{attribute addProperty BoxType "APS1003-5000-0016"}
{attribute addProperty Id "FB_InputsAT %I*FB_Inputs_245CD1AC24643080WcStateAT %I*WcState_F855686C1620InfoDataAT %I*InfoData_7231B2DD80100"}
{attribute addProperty CRC "3520049983"}
{attribute addProperty SizeInBites "2560"}
{attribute addProperty SizeInBytes "320"}
TYPE APS1003_147A8693 :
STRUCT
	{attribute addProperty Name "FB_Inputs"}
	FB_Inputs : FB_Inputs_245CD1AC;
	{attribute addProperty Name "WcState"}
	WcState : WcState_F855686C;
	{attribute addProperty Name "InfoData"}
	InfoData : InfoData_7231B2DD;
END_STRUCT
END_TYPE

(* stored: Version 1.2.0.0, ProductVersion 3.1.4024.9
   DUT APS1003_147A8693: Id {9d30afb5-31c9-4b7f-9a48-0bbdb881849f} *)
